// TIA Portal V16 export
// export: Created 2024-12-03T15:41:46.288835Z, ExportSetting WithReadOnly, DisplayName Totally Integrated Automation Portal, DisplayVersion V16 Update 6, DisplayName TIA Portal Version Control Interface, DisplayVersion V16 Update 2, DisplayName TIA Portal Openness, DisplayVersion V16 Update 6, DisplayName TIA Portal Teamcenter Gateway, DisplayVersion V16, DisplayName SINAMICS Startdrive Advanced, DisplayVersion V16 Update 5, DisplayName SINAMICS Startdrive G130, G150, S120, S150, SINAMICS MV, S210, DisplayVersion V16 Update 5, DisplayName SINAMICS Startdrive G110M, G120, G120C, G120D, G120P, G115D, DisplayVersion V16 Update 5, DisplayName STEP 7 Professional, DisplayVersion V16 Update 6, DisplayName STEP 7 Safety, DisplayVersion V16, DisplayName WinCC Advanced / Unified PC, DisplayVersion V16 Update 6
TYPE "IPC_INTERFACE_STATUS_UDT"
// stored: CreationDate 2021-07-13T07:41:36.2278727Z, InterfaceModifiedDate 2021-06-24T07:26:07.648876Z, IsConsistent true, LibraryConformanceStatus The object is library-conformant., ModifiedDate 2021-06-24T07:26:07.648876Z
   STRUCT
      Diagnostics : Struct
         TimeOuts : DInt;
         Successes : DInt;
         OutOfSync : DInt;
         CommunicationTime : Time;
         LastCommunicationTime : Time;
      END_STRUCT;
      ResultStatus : Struct
         static : "IPC_RES_STATUS_UDT";
         pulse : "IPC_RES_STATUS_UDT";
      END_STRUCT;
      Status : Struct
         online : Bool;
         ReadyForSendingData : Bool;
         ReceivingData : Bool;
      END_STRUCT;
      Settings : Struct
         TimeOut : Time := t#1s;
         RetrySending : Bool;
         RetryThreshold : Int;
         RetryCounter : Int := 0;
         ResendMessage : Time := t#1s;   // The time when the object will execute a retry
      END_STRUCT;
      Zone { S7_SetPoint := 'True'} : UInt;
      "name" : String[20];
   END_STRUCT;
END_TYPE
